// TIA Portal project "Bombas" (V17)

(* hardware
DEVICE "S7-1500/ET200MP station_1"  S7-1500 station
   slot 0: "Rail_0"  Rack  6ES7 590-1***0-0AA0
   slot 1: "PLC_1"  CPU 1511-1 PN  6ES7 511-1AK00-0AB0  V1.8
      slot 3: "CPU display_1"  6ES7591-1AA00-0AA0
      slot 32768: "PROFINET interface_1"  X1
         slot 32769: "Port_1"  X1 P1
         slot 32770: "Port_2"  X1 P2
*)

// ===== PLC "PLC_1"  CPU 1511-1 PN =====

VAR_GLOBAL   // PLC tag table "Default tag table"
   "A" AT %I0.0 : Bool;
   "P" AT %I0.1 : Bool;
   "NB_T1" AT %I0.2 : Bool;
   "NA_T1" AT %I0.3 : Bool;
   "NB_P1" AT %I0.4 : Bool;
   "NA_P1" AT %I0.5 : Bool;
   "SC1_S1" AT %I0.6 : Bool;
   "SC2_S1" AT %I0.7 : Bool;
   "NB_T2" AT %I1.0 : Bool;
   "NA_T2" AT %I1.1 : Bool;
   "NB_P2" AT %I1.2 : Bool;
   "NA_P2" AT %I1.3 : Bool;
   "SC1_S2" AT %I1.4 : Bool;
   "SC2_S2" AT %I1.5 : Bool;
   "NB_T3" AT %I1.6 : Bool;
   "NA_T3" AT %I1.7 : Bool;
   "NB_P3" AT %I2.0 : Bool;
   "NA_P3" AT %I2.1 : Bool;
   "SC1_S3" AT %I2.2 : Bool;
   "SC2_S3" AT %I2.3 : Bool;
   "B1_S1" AT %Q0.0 : Bool;
   "B2_S1" AT %Q0.1 : Bool;
   "B1_S2" AT %Q0.2 : Bool;
   "B2_S2" AT %Q0.3 : Bool;
   "B1_S3" AT %Q0.4 : Bool;
   "B2_S3" AT %Q0.5 : Bool;
END_VAR

DATA_BLOCK "SUBSYS_DB"   // DB1
{ S7_Optimized_Access := 'TRUE' }
VERSION : 0.1
// stored: InstanceOfName SUBSYS
"SUBSYS"
BEGIN
END_DATA_BLOCK

DATA_BLOCK "SUBSYS_DB_1"   // DB2
{ S7_Optimized_Access := 'TRUE' }
VERSION : 0.1
// stored: InstanceOfName SUBSYS
"SUBSYS"
BEGIN
END_DATA_BLOCK

DATA_BLOCK "SUBSYS_DB_2"   // DB3
{ S7_Optimized_Access := 'TRUE' }
VERSION : 0.1
// stored: InstanceOfName SUBSYS
"SUBSYS"
BEGIN
END_DATA_BLOCK

DATA_BLOCK "MANAGER_DB"   // DB4
{ S7_Optimized_Access := 'TRUE' }
VERSION : 0.1
// stored: InstanceOfName MANAGER
"MANAGER"
BEGIN
END_DATA_BLOCK

FUNCTION_BLOCK "SUBSYS"   // FB1, GRAPH_PLUS
{ S7_Optimized_Access := 'TRUE' }
VERSION : 0.1
   VAR_INPUT
      ACK_EF : Bool := false;   // Acknowledge all errors and faults
      "NB_T#" : Bool;
      "NA_T#" : Bool;
      "NB_P#" : Bool;
      "NA_P#" : Bool;
   END_VAR
   VAR_OUTPUT
      "B1_S#" : Bool;
      "B2_S#" : Bool;
   END_VAR
   VAR
      HMI_INFO : Array[0..8] of UInt;
      IF_PAR : G7_IfParPlus_V2;
      RT_DATA : G7_RTDataPlus_V2;   // Internal data area
      Trans1 : G7_TransitionPlus_V2;   // Transition structure
      Trans2 : G7_TransitionPlus_V2;   // Transition structure
      Trans3 : G7_TransitionPlus_V2;   // Transition structure
      Trans4 : G7_TransitionPlus_V2;   // Transition structure
      Step1 : G7_StepPlus_V2;   // Step structure
      Step2 : G7_StepPlus_V2;   // Step structure
      Step3 : G7_StepPlus_V2;   // Step structure
      Step4 : G7_StepPlus_V2;   // Step structure
      SINI : Array[0..1] of USInt;
      LSTT : Array[0..3] of USInt;
      ATAJ : Array[0..3] of USInt;
      ATAB : Array[0..3] of USInt;
      PSTT : Array[0..3] of USInt;
      NSTT : Array[0..3] of USInt;
      ASSJ : Array[0..3] of USInt;
      ASSB : Array[0..3] of USInt;
      PTTS : Array[0..3] of USInt;
      NTTS : Array[0..3] of USInt;
      SW_SQTS : Array[0..3] of USInt;
      SWITCH : Array[0..0] of USInt;
      TVX : Array[0..1] of USInt;
      TTX : Array[0..1] of USInt;
      TSX : Array[0..1] of USInt;
      S00X : Array[0..1] of USInt;
      SOFFX : Array[0..1] of USInt;
      SONX : Array[0..1] of USInt;
      SAX : Array[0..1] of USInt;
      SERRX : Array[0..4] of USInt;
      SMX : Array[0..4] of USInt;
      S0X : Array[0..4] of USInt;
      S1X : Array[0..4] of USInt;
      IL_ALARM_INST : Program_Alarm;
      SUP_ALARM_INST : Program_Alarm;
      STEP_TIME_ALARM_INST : Program_Alarm;
      IEC_TIMER_INST : IEC_TIMER;
      TRANSACTION_FLAG : Bool := false;
   END_VAR
   // SINI[0] := 2;
   // LSTT[0] := 255;
   // LSTT[1] := 255;
   // LSTT[2] := 255;
   // ATAJ[1] := 1;
   // ATAJ[2] := 2;
   // ATAJ[3] := 3;
   // ATAB[1] := 1;
   // ATAB[2] := 2;
   // ATAB[3] := 3;
   // PSTT[1] := 1;
   // PSTT[2] := 2;
   // PSTT[3] := 3;
   // NSTT[0] := 1;
   // NSTT[1] := 2;
   // NSTT[2] := 3;
   // ASSJ[1] := 1;
   // ASSJ[2] := 2;
   // ASSJ[3] := 3;
   // ASSB[1] := 1;
   // ASSB[2] := 2;
   // ASSB[3] := 3;
   // PTTS[0] := 255;
   // PTTS[2] := 1;
   // PTTS[3] := 2;
   // NTTS[1] := 1;
   // NTTS[2] := 2;
   // NTTS[3] := 3;
   // TVX[0] := 16#1;
   // TTX[0] := 16#1;
   // TSX[0] := 16#1;
   // S00X[0] := 16#1;
   // SOFFX[0] := 16#1;
   // SONX[0] := 16#1;
   // SAX[0] := 16#1;
   // SERRX[0] := 16#1;
   // SMX[0] := 16#1;
   // S0X[0] := 16#1;
   // S1X[0] := 16#1;
BEGIN
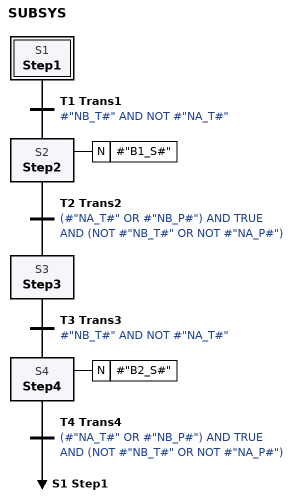
   // sequencer 1
   INITIAL_STEP Step1:   // S1, max time T#10S, warning time T#7S
   END_STEP
   TRANSITION Trans1 FROM Step1 TO Step2   // T1
      := #"NB_T#" AND NOT #"NA_T#";
   END_TRANSITION
   STEP Step2:   // S2, max time T#10S, warning time T#7S
              N    #"B1_S#"
   END_STEP
   TRANSITION Trans2 FROM Step2 TO Step3   // T2
      := (#"NA_T#" OR #"NB_P#") AND TRUE AND (NOT #"NB_T#" OR NOT #"NA_P#");
   END_TRANSITION
   STEP Step3:   // S3, max time T#10S, warning time T#7S
   END_STEP
   TRANSITION Trans3 FROM Step3 TO Step4   // T3
      := #"NB_T#" AND NOT #"NA_T#";
   END_TRANSITION
   STEP Step4:   // S4, max time T#10S, warning time T#7S
              N    #"B2_S#"
   END_STEP
   TRANSITION Trans4 FROM Step4 TO Step1   // T4, jump
      := (#"NA_T#" OR #"NB_P#") AND TRUE AND (NOT #"NB_T#" OR NOT #"NA_P#");
   END_TRANSITION
END_FUNCTION_BLOCK

FUNCTION_BLOCK "MANAGER"   // FB2, GRAPH_PLUS
{ S7_Optimized_Access := 'TRUE' }
VERSION : 0.1
   VAR_INPUT
      P : Bool;
      "A" : Bool;
      SC1_S3 : Bool;
      SC2_S3 : Bool;
      SC2_S2 : Bool;
      SC1_S2 : Bool;
      SC1_S1 : Bool;
      SC2_S1 : Bool;
      NA_T1 : Bool;
      NB_T1 : Bool;
      NA_P1 : Bool;
      NB_P1 : Bool;
      NA_T2 : Bool;
      NB_T2 : Bool;
      NA_P2 : Bool;
      NB_P2 : Bool;
      NA_T3 : Bool;
      NB_T3 : Bool;
      NA_P3 : Bool;
      ACK_EF : Bool := false;   // Acknowledge all errors and faults
      NB_P3 : Bool;
   END_VAR
   VAR_OUTPUT
      B2_S3 : Bool;
      B1_S3 : Bool;
      B2_S2 : Bool;
      B1_S2 : Bool;
      B2_S1 : Bool;
      B1_S1 : Bool;
   END_VAR
   VAR
      HMI_INFO : Array[0..11] of UInt;
      IF_PAR : G7_IfParPlus_V2;
      RT_DATA : G7_RTDataPlus_V2;   // Internal data area
      Trans1 : G7_TransitionPlus_V2;   // Transition structure
      Trans2 : G7_TransitionPlus_V2;   // Transition structure
      Trans3 : G7_TransitionPlus_V2;   // Transition structure
      Trans4 : G7_TransitionPlus_V2;   // Transition structure
      Trans5 : G7_TransitionPlus_V2;   // Transition structure
      Step1 : G7_StepPlus_V2;   // Step structure
      Step2 : G7_StepPlus_V2;   // Step structure
      Step3 : G7_StepPlus_V2;   // Step structure
      Step4 : G7_StepPlus_V2;   // Step structure
      Step5 : G7_StepPlus_V2;   // Step structure
      Step6 : G7_StepPlus_V2;   // Step structure
      Step7 : G7_StepPlus_V2;   // Step structure
      SINI : Array[0..4] of USInt;
      LSTT : Array[0..4] of USInt;
      ATAJ : Array[0..4] of USInt;
      ATAB : Array[0..4] of USInt;
      PSTT : Array[0..4] of USInt;
      NSTT : Array[0..4] of USInt;
      ASSJ : Array[0..6] of USInt;
      ASSB : Array[0..6] of USInt;
      PTTS : Array[0..6] of USInt;
      NTTS : Array[0..6] of USInt;
      SW_SQTS : Array[0..6] of USInt;
      SWITCH : Array[0..1] of USInt;
      TVX : Array[0..4] of USInt;
      TTX : Array[0..4] of USInt;
      TSX : Array[0..4] of USInt;
      S00X : Array[0..4] of USInt;
      SOFFX : Array[0..4] of USInt;
      SONX : Array[0..4] of USInt;
      SAX : Array[0..4] of USInt;
      SERRX : Array[0..7] of USInt;
      SMX : Array[0..7] of USInt;
      S0X : Array[0..7] of USInt;
      S1X : Array[0..7] of USInt;
      IL_ALARM_INST : Program_Alarm;
      SUP_ALARM_INST : Program_Alarm;
      STEP_TIME_ALARM_INST : Program_Alarm;
      IEC_TIMER_INST : IEC_TIMER;
      TRANSACTION_FLAG : Bool := false;
   END_VAR
   // SINI[0] := 2;
   // SINI[2] := 255;
   // SINI[3] := 255;
   // SINI[4] := 255;
   // LSTT[0] := 255;
   // LSTT[2] := 255;
   // LSTT[3] := 255;
   // LSTT[4] := 255;
   // ATAJ[1] := 1;
   // ATAJ[2] := 2;
   // ATAJ[3] := 3;
   // ATAJ[4] := 4;
   // ATAB[1] := 1;
   // ATAB[2] := 2;
   // ATAB[3] := 3;
   // ATAB[4] := 4;
   // PSTT[1] := 4;
   // PSTT[2] := 1;
   // PSTT[3] := 3;
   // PSTT[4] := 2;
   // NSTT[0] := 1;
   // NSTT[2] := 4;
   // NSTT[3] := 5;
   // NSTT[4] := 6;
   // ASSJ[1] := 1;
   // ASSJ[2] := 2;
   // ASSJ[3] := 3;
   // ASSJ[4] := 5;
   // ASSJ[5] := 6;
   // ASSJ[6] := 4;
   // ASSB[1] := 3;
   // ASSB[2] := 1;
   // ASSB[3] := 2;
   // ASSB[4] := 4;
   // ASSB[5] := 5;
   // ASSB[6] := 6;
   // PTTS[0] := 255;
   // PTTS[4] := 2;
   // PTTS[5] := 3;
   // PTTS[6] := 4;
   // NTTS[1] := 2;
   // NTTS[2] := 4;
   // NTTS[3] := 3;
   // NTTS[4] := 1;
   // NTTS[5] := 1;
   // NTTS[6] := 1;
   // SW_SQTS[1] := 1;
   // SW_SQTS[2] := 2;
   // SW_SQTS[3] := 3;
   // SW_SQTS[4] := 1;
   // SW_SQTS[5] := 3;
   // SW_SQTS[6] := 2;
   // SWITCH[0] := 192;
   // SWITCH[1] := 106;
   // TVX[0] := 16#1;
   // TTX[0] := 16#1;
   // TSX[0] := 16#1;
   // S00X[0] := 16#1;
   // SOFFX[0] := 16#1;
   // SONX[0] := 16#1;
   // SAX[0] := 16#1;
   // SERRX[0] := 16#1;
   // SMX[0] := 16#1;
   // S0X[0] := 16#1;
   // S1X[0] := 16#1;
BEGIN
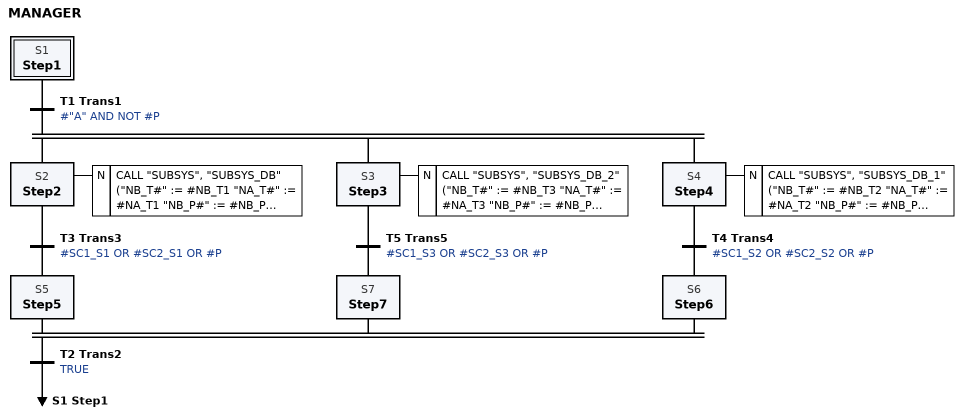
   // sequencer 1
   INITIAL_STEP Step1:   // S1, max time T#10S, warning time T#7S
   END_STEP
   TRANSITION Trans1 FROM Step1 TO (Step2, Step3, Step4)   // T1
      := #"A" AND NOT #P;
   END_TRANSITION
   STEP Step2:   // S2, max time T#10S, warning time T#7S
              N    CALL "SUBSYS", "SUBSYS_DB"
                   ("NB_T#" := #NB_T1
                   "NA_T#" := #NA_T1
                   "NB_P#" := #NB_P1
                   "NA_P#" := #NA_P1
                   "B1_S#" => #B1_S1
                   "B2_S#" => #B2_S1
                   )
   END_STEP
   TRANSITION Trans3 FROM Step2 TO Step5   // T3
      := #SC1_S1 OR #SC2_S1 OR #P;
   END_TRANSITION
   STEP Step3:   // S3, max time T#10S, warning time T#7S
              N    CALL "SUBSYS", "SUBSYS_DB_2"
                   ("NB_T#" := #NB_T3
                   "NA_T#" := #NA_T3
                   "NB_P#" := #NB_P3
                   "NA_P#" := #NA_P3
                   "B1_S#" => #B1_S3
                   "B2_S#" => #B2_S3
                   )
   END_STEP
   TRANSITION Trans5 FROM Step3 TO Step7   // T5
      := #SC1_S3 OR #SC2_S3 OR #P;
   END_TRANSITION
   STEP Step4:   // S4, max time T#10S, warning time T#7S
              N    CALL "SUBSYS", "SUBSYS_DB_1"
                   ("NB_T#" := #NB_T2
                   "NA_T#" := #NA_T2
                   "NB_P#" := #NB_P2
                   "NA_P#" := #NA_P2
                   "B1_S#" => #B1_S2
                   "B2_S#" => #B2_S2
                   )
   END_STEP
   TRANSITION Trans4 FROM Step4 TO Step6   // T4
      := #SC1_S2 OR #SC2_S2 OR #P;
   END_TRANSITION
   STEP Step5:   // S5, max time T#10S, warning time T#7S
   END_STEP
   STEP Step6:   // S6, max time T#10S, warning time T#7S
   END_STEP
   STEP Step7:   // S7, max time T#10S, warning time T#7S
   END_STEP
   TRANSITION Trans2 FROM (Step5, Step6, Step7) TO Step1   // T2, jump
      := TRUE;
   END_TRANSITION
END_FUNCTION_BLOCK

ORGANIZATION_BLOCK "Main"   // OB1, LAD, ProgramCycle
TITLE = "Main Program Sweep (Cycle)"
{ S7_Optimized_Access := 'TRUE' }
VERSION : 0.1
   VAR_INPUT
      Initial_Call : Bool;   // Initial call of this OB
      Remanence : Bool;   // =True, if remanent data are available
   END_VAR
BEGIN

REGION Network 1
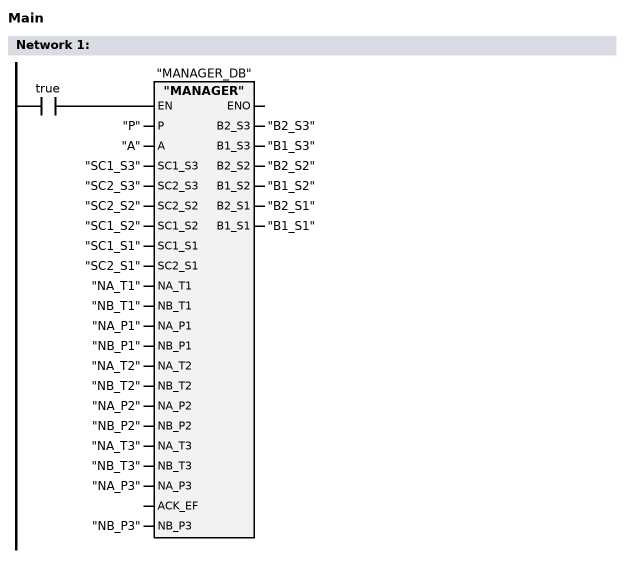
   RUNG wire#powerrail
      Contact( true )
      "MANAGER_DB"(P := "P", "A" := "A", SC1_S3 := "SC1_S3", SC2_S3 := "SC2_S3", SC2_S2 := "SC2_S2", SC1_S2 := "SC1_S2", SC1_S1 := "SC1_S1", SC2_S1 := "SC2_S1", NA_T1 := "NA_T1", NB_T1 := "NB_T1", NA_P1 := "NA_P1", NB_P1 := "NB_P1", NA_T2 := "NA_T2", NB_T2 := "NB_T2", NA_P2 := "NA_P2", NB_P2 := "NB_P2", NA_T3 := "NA_T3", NB_T3 := "NB_T3", NA_P3 := "NA_P3", ACK_EF :=, NB_P3 := "NB_P3", B2_S3 => "B2_S3", B1_S3 => "B1_S3", B2_S2 => "B2_S2", B1_S2 => "B1_S2", B2_S1 => "B2_S1", B1_S1 => "B1_S1")
   END_RUNG
   // the same network as SCL:
   IF true THEN
       "MANAGER_DB"(P := "P",   // "MANAGER"
                    "A" := "A",
                    SC1_S3 := "SC1_S3",
                    SC2_S3 := "SC2_S3",
                    SC2_S2 := "SC2_S2",
                    SC1_S2 := "SC1_S2",
                    SC1_S1 := "SC1_S1",
                    SC2_S1 := "SC2_S1",
                    NA_T1 := "NA_T1",
                    NB_T1 := "NB_T1",
                    NA_P1 := "NA_P1",
                    NB_P1 := "NB_P1",
                    NA_T2 := "NA_T2",
                    NB_T2 := "NB_T2",
                    NA_P2 := "NA_P2",
                    NB_P2 := "NB_P2",
                    NA_T3 := "NA_T3",
                    NB_T3 := "NB_T3",
                    NA_P3 := "NA_P3",
                    NB_P3 := "NB_P3",
                    B2_S3 => "B2_S3",
                    B1_S3 => "B1_S3",
                    B2_S2 => "B2_S2",
                    B1_S2 => "B1_S2",
                    B2_S1 => "B2_S1",
                    B1_S1 => "B1_S1");
   END_IF;
END_REGION
END_ORGANIZATION_BLOCK